{attribute 'no_explicit_call' := 'Direct call is not allowed'} 
FUNCTION_BLOCK StringBuilder EXTENDS Object
VAR CONSTANT
	STRING_CHAR_SIZE : BYTE := 1;
END_VAR
VAR
	_ClassName : STRING := __POUNAME();

	_String : POINTER TO STRING;
	_Length : UDINT;
	_Capacity : UDINT;
END_VAR

METHOD Append : REFERENCE TO StringBuilder
VAR_INPUT
	value : ANY;
END_VAR
InternalAppend(value);

Append REF= THIS^;
END_METHOD

METHOD AppendIf : REFERENCE TO StringBuilder
VAR_INPUT
	value : ANY;
	condition : BOOL;
END_VAR
IF condition THEN
	InternalAppend(value);
END_IF

AppendIf REF= THIS^;
END_METHOD

METHOD AppendString : REFERENCE TO StringBuilder
VAR_IN_OUT CONSTANT
	value : STRING;
END_VAR
VAR
	valueDescriptor : __SYSTEM.AnyType;
END_VAR
valueDescriptor.TypeClass := __SYSTEM.TYPE_CLASS.TYPE_STRING;
valueDescriptor.pValue := ADR(value);
valueDescriptor.diSize := TO_DINT(Tc2_Utilities.LEN2(ADR(value))) + 1;

InternalAppend(valueDescriptor);

AppendString REF= THIS^;
END_METHOD

METHOD AppendStringIf : REFERENCE TO StringBuilder
VAR_IN_OUT CONSTANT
	value : STRING;
END_VAR
VAR_INPUT
	condition : BOOL;
END_VAR
VAR
	valueDescriptor : __SYSTEM.AnyType;
END_VAR
IF condition THEN
	valueDescriptor.TypeClass := __SYSTEM.TYPE_CLASS.TYPE_STRING;
	valueDescriptor.pValue := ADR(value);
	valueDescriptor.diSize := TO_DINT(Tc2_Utilities.LEN2(ADR(value))) + 1;
	
	InternalAppend(valueDescriptor);
END_IF

AppendStringIf REF= THIS^;
END_METHOD

METHOD AssignToString : BOOL
VAR_INPUT
	targetString : ANY_STRING;
END_VAR
VAR
	//exceptionFactory : ExceptionFactory(__POUNAME(), ClassName, CurrentNamespace.Name);
END_VAR
IF targetString.TypeClass <> __SYSTEM.TYPE_CLASS.TYPE_STRING THEN
	//exceptionFactory.ThrowException(__POSITION(), "Invalid string type, should be STRING");
END_IF

IF targetString.diSize < TO_DINT(_Length + STRING_CHAR_SIZE) THEN
	//exceptionFactory.ThrowException(__POSITION(), WStringHelper.Concat5("Target string size is ", TO_WSTRING(targetString.diSize), " bytes, but built string is ", TO_WSTRING(_Length + STRING_CHAR_SIZE), " bytes"));
END_IF

AssignToString := Tc2_Utilities.STRNCPY(targetString.pValue, _String, TO_UDINT(targetString.diSize));
END_METHOD

PROPERTY Capacity : UDINT
GET
Capacity := _Capacity;
END_GET
END_PROPERTY

{attribute 'monitoring' := 'call'}
PROPERTY ClassName : STRING
GET
ClassName := _ClassName;
END_GET
END_PROPERTY

METHOD Clear : REFERENCE TO StringBuilder
VAR_INPUT
	releaseMemory : BOOL;
END_VAR
_Length := 0;

IF _Capacity > 0 THEN
	IF releaseMemory THEN
		__DELETE(_String);	
		_Capacity := 0;	
	ELSE
		Tc2_System.MEMSET(_String, 0, StringMaxSize);
	END_IF	
END_IF

Clear REF= THIS^;
END_METHOD

METHOD ClearIf : REFERENCE TO StringBuilder
VAR_INPUT
	condition : BOOL;
	releaseMemory : BOOL;
END_VAR
IF condition THEN
	Clear(releaseMemory);
END_IF

ClearIf REF= THIS^;
END_METHOD

METHOD FB_exit : BOOL
VAR_INPUT
	bInCopyCode : BOOL; // if TRUE, the exit method is called for exiting an instance that is copied afterwards (online change).
END_VAR
Clear(TRUE);
END_METHOD

METHOD PROTECTED InternalAppend 
VAR_INPUT
	value : REFERENCE TO __System.AnyType;
END_VAR
VAR
	stringToAppend : STRING(255);	
	stringToAppendLength : UDINT;
	newString : POINTER TO BYTE;
	newCapacity : UDINT;
END_VAR
stringToAppend := StringHelper.InternalAnyToString(value);

stringToAppendLength := TO_UDINT(Tc2_Standard.LEN(stringToAppend));

IF _Capacity = 0 OR_ELSE _Length + stringToAppendLength > _Capacity THEN
	IF _Length + stringToAppendLength - _Capacity > 80 THEN
		newCapacity := _Length + stringToAppendLength;
	ELSE
		newCapacity := _Length + 80;
	END_IF
	
	newString := __NEW(BYTE, (STRING_CHAR_SIZE + (newCapacity * STRING_CHAR_SIZE)));
	
	IF _String <> 0 THEN
		Tc2_Utilities.STRNCPY(newString, _String, STRING_CHAR_SIZE + (newCapacity * STRING_CHAR_SIZE));
		
		__DELETE(_String);
	END_IF
	
	_String := newString;
	_Capacity := newCapacity;
END_IF

Tc2_Utilities.CONCAT2(_String, ADR(stringToAppend), _String, StringMaxSize);
_Length := _Length + stringToAppendLength;
END_METHOD

PROPERTY StringAddress : POINTER TO STRING
GET
StringAddress := _String;
END_GET
END_PROPERTY

PROPERTY StringLength : UDINT
GET
StringLength := _Length;
END_GET
END_PROPERTY

PROPERTY StringMaxSize : UDINT
GET
StringMaxSize := STRING_CHAR_SIZE + (STRING_CHAR_SIZE * _Capacity);
END_GET
END_PROPERTY

PROPERTY StringRealSize : UDINT
GET
StringRealSize := STRING_CHAR_SIZE + (STRING_CHAR_SIZE * _Length);
END_GET
END_PROPERTY

METHOD ToString255 : STRING(255)
IF _Length > 0 THEN
	Tc2_Utilities.STRNCPY(ADR(ToString255), _String, SIZEOF(ToString255));
END_IF
END_METHOD

END_FUNCTION_BLOCK

(* stored: Version 1.1.0.1
   POU StringBuilder: Id {f03c5ece-54b0-49bc-9e74-735ce698ca91}, SpecialFunc None
   Folder Service members: Id {968318cb-c8ed-4cd3-be47-9ebc32f63088}
   Method Append: Id {dabe62c3-04fc-470c-be60-55b4ed188ae0}
   Method AppendIf: Id {199dc18c-dbee-4779-9a13-c1714bd95dcf}
   Method AppendString: Id {c666509b-6bf8-4c72-8b5e-b19bc686e00f}
   Method AppendStringIf: Id {074a9d5c-1674-41db-9481-836536b59c02}
   Method AssignToString: Id {10d5f0e9-9271-4cc3-8d0d-dfdcab9d69d7}
   Property Capacity: Id {f8fe2243-a830-43e2-ac65-94c2bac2e83b}
   Get Get: Id {2dcab30d-891f-4012-bbc4-3c011458bd6c}
   Property ClassName: Id {96c5f4ec-8cc2-45ef-9959-bf29c92c37f2}
   Get Get: Id {f5e2c5d7-95d2-413b-81d4-e7080afffeed}
   Method Clear: Id {8f5522b9-3d81-4242-abd7-dd4273b2b25a}
   Method ClearIf: Id {d2833228-db47-4f2b-8573-13851a05bb46}
   Method FB_exit: Id {12ceaea3-1041-4d55-a8ca-67665e1a171d}
   Method InternalAppend: Id {0070b123-ec19-4046-98c8-fe14f169788e}
   Property StringAddress: Id {2d1338d4-5f7d-449c-9eb8-4e1a567e1527}
   Get Get: Id {926d0cb4-b86d-4e38-ab52-0ec7140a7f9c}
   Property StringLength: Id {a9741d45-bf3c-474a-bc1f-6e40d481d113}
   Get Get: Id {1fd67579-9713-4351-8721-ed4f49a9ddab}
   Property StringMaxSize: Id {04271010-02b5-471f-a68d-cda3e502098a}
   Get Get: Id {881ff8bf-4670-40a5-85d5-b0f10c02707b}
   Property StringRealSize: Id {85c7974d-7e7c-44a4-b392-d52ee514e0e4}
   Get Get: Id {384b73a5-42c9-44f4-a6fd-5da5289cf624}
   Method ToString255: Id {d06c15ee-6eaf-4994-b132-31a1ad6c58ba} *)
